(* Logix 5000 project; controller EuniceF_ICA12 vendor 1 type 14 code 150 rev 37.11; software revision 37.00 *)

TASK MainTask (continuous, watchdog 500 ms) : MainProgram

MODULES
   Local : vendor 1 type 14 code 150 (Compact 0, rev 37.11)
      Discrete_IO : Embedded (Compact 1, rev 3.1, Output RPI 20 ms)
      Analog_IO : Embedded (Compact 2, rev 1.1, Output RPI 80 ms)
      Counters : Embedded (Compact 3, rev 1.1, Output RPI 20 ms)
END_MODULES

VAR_GLOBAL   (* controller tags *)
   MOTOR : ALIAS FOR Local:1:O.Data.1;
   MOTOR1 : ALIAS FOR Local:1:O.Data.1;
   MOTOR2 : ALIAS FOR Local:1:O.Data.2;
   MOTOR3 : ALIAS FOR Local:1:O.Data.3;
   START : ALIAS FOR Local:1:I.Data.11;
   STOP : ALIAS FOR Local:1:I.Data.8;
   Timer1 : TIMER := (PRE := 5000);
   TIMER2 : TIMER := (PRE := 3000);
END_VAR

PROGRAM MainProgram   (* main routine MainRoutine *)

ROUTINE MainRoutine   (* ladder *)
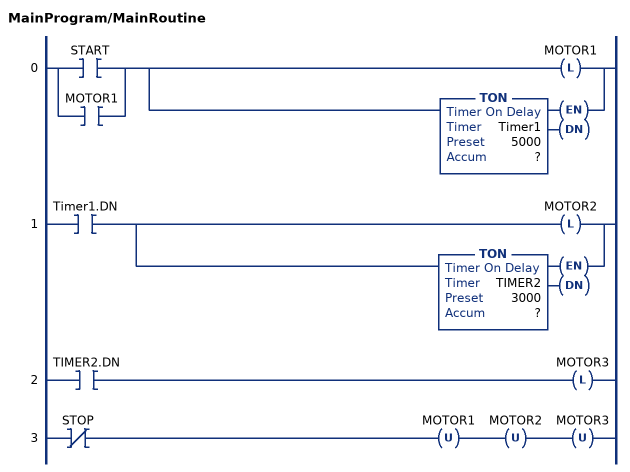
   0: [XIC(START) ,XIC(MOTOR1) ][OTL(MOTOR1) ,TON(Timer1,?,?) ];
   1: XIC(Timer1.DN)[OTL(MOTOR2) ,TON(TIMER2,?,?) ];
   2: XIC(TIMER2.DN)OTL(MOTOR3);
   3: XIO(STOP)OTU(MOTOR1)OTU(MOTOR2)OTU(MOTOR3);
END_ROUTINE
END_PROGRAM
